(*
  This fb handles mechanical print unit corrections.
  - a 4p grid distortion
  - print unit bar banana correction
  NOTE: temperature extention of whole printbar is still handled in camera
*)
FUNCTION_BLOCK FB_FineAlignement EXTENDS FB_BasePrint IMPLEMENTS I_GridPointCorrection
VAR
  // config
  _fPxResolution     : LREAL; // pixel resolution

  // corrections
  //-- 4 point PU deformation correction/distortion
  //    VISU setup point providing reference and correction (NOTE: persists settings internally)
  _fbPUCorrPoints    : ARRAY[1..4] OF FB_PointCorr;
  //-- banana correction
  _fT1 : LREAL;   // temperature 1
  _fT2 : LREAL;   // temperature 2
  _dx_middle : LREAL;  // correction in middle (for view only)
  _y_max : LREAL; // print unit width [mm]
  //-- PUC 4p correction
  _pAdsCam           : POINTER TO FB_ADS_CAMERA;  // camera interface PUC
  aPucPointNames : ARRAY[1..4] OF STRING := ['1 blue','2 red','3 green','4 olive'];
  
  // helper
  lCtr     : UDINT;
  
  // unit test & debug
  _bUT_4p, _bUT_banana, _bUT_4pPuc : BOOL;
  _sUTPoints_dx : ARRAY[0..nC_UT_cols, 0..nC_UT_rows] OF LREAL;
  _sUTPoints_dy : ARRAY[0..nC_UT_cols, 0..nC_UT_rows] OF LREAL;
  // 4pPUC
  bSelect : ARRAY[1..4] OF BOOL;
  bSelected : ARRAY[1..4] OF BOOL;
  bXPlus, bXMinus, bYPlus, bYMinus : BOOL;
  bTest4pPuc_running : BOOL;
END_VAR
VAR PERSISTENT
  //-- 4point correction
  _bEnable_4p    : BOOL := FALSE;
  _bEnablePuc_4p : BOOL := FALSE;
  //  persistence of points see: FB_PointCorr
  //-- banana correction
  _bEnable_banana : BOOL := FALSE;
  _e_max_per_deltaT : LREAL := 0.01;  // [mm/°C]  TODO: use from config
END_VAR
VAR CONSTANT
  // Unit test configuration
  nC_UT_cols : DINT := 6;   // for test only
  nC_UT_rows : DINT := 5;   // for test only
END_VAR

// cyclic caluclation and view updates
//        NOTE: deformation is happening in updateCorrection() callback

//-- 4p correction
//   visu overrides (limitation rectancular point definition)
_fbPUCorrPoints[3].fX_Ref := _fbPUCorrPoints[1].fX_Ref;
_fbPUCorrPoints[4].fX_Ref := _fbPUCorrPoints[2].fX_Ref;
_fbPUCorrPoints[2].fY_Ref := _fbPUCorrPoints[1].fY_Ref;
_fbPUCorrPoints[4].fY_Ref := _fbPUCorrPoints[3].fY_Ref;
//   update CorrectionPoints view elements
FOR lCtr := 1 TO 4 DO
  _fbPUCorrPoints[lCtr](); 
END_FOR

//-- banana correction
// just calculate the dx in the middle of the PU, just for the VISU
calc_banana_correction(x_pos:=0, y_pos:=_y_max/(2*1000), fT1:=_fT1, fT2:=_fT2, dx_corr=>_dx_middle);
_dx_middle := _dx_middle * 1000; // [m] --> [mm] for visu

// Unit test
IF _bUT_4p THEN _bUT_4p := FALSE; _test_4p(); END_IF
IF _bUT_banana THEN _bUT_banana := FALSE; _test_banana(); END_IF
IF _bUT_4pPuc THEN _test_Puc4p(); END_IF

METHOD PRIVATE _test_4p
VAR
  sPoint : ST_DeformationPoint;
  nCol, nRow, nCrPoint : DINT;
  dx, dy : LREAL;       // correction in [m]
  dx_px, dy_px : DINT;  // correction in [px]
  pPUC_CorrPointsInd : POINTER TO ARRAY[1..4] OF ST_CORRECTION_POINT;
  
  nCorrectionX : ARRAY[1..4] OF REAL := [-0.25, -0.2, 0.35, 0.35];
  nCorrectionY : ARRAY[1..4] OF REAL := [-0.45, -0.3, -0.8, -0.65];
  nCorrectionPointX_PLC : ARRAY[1..4] OF REAL := [0, 1000,   0, 1000];
  nCorrectionPointY_PLC : ARRAY[1..4] OF REAL := [0,   0, 702, 702];
  nCorrectionPointX_PUC : ARRAY[1..4] OF REAL := [0, 671.99,   0, 671.99];
  nCorrectionPointY_PUC : ARRAY[1..4] OF REAL := [-0.0001666666, -0.0001666666, 754.2108, 754.2108];
END_VAR
// setup test correcton points location for PLC & PUC 4p testing
pPUC_CorrPointsInd := _pAdsCam^.pCorrectionPointsIndication;
IF pPUC_CorrPointsInd = 0 THEN F_Report_Error(ErrType:=EN_REPORT_ERROR_TYPE.Report_Error_0Pointer);  RETURN; END_IF

FOR nCrPoint:=1 TO 4 DO
  // correction point location
  // -- PLC
  _fbPUCorrPoints[nCrPoint].fX_Ref := nCorrectionPointX_PLC[nCrPoint];
  _fbPUCorrPoints[nCrPoint].fY_Ref := nCorrectionPointY_PLC[nCrPoint];
  // -- PUC  
  pPUC_CorrPointsInd^[nCrPoint].posx := nCorrectionPointX_PUC[nCrPoint];
  pPUC_CorrPointsInd^[nCrPoint].posy := nCorrectionPointY_PUC[nCrPoint];
  
  // point correction  
  // -- PLC
  _fbPUCorrPoints[nCrPoint].fX := nCorrectionX[nCrPoint];
  _fbPUCorrPoints[nCrPoint].fY := nCorrectionY[nCrPoint];
  // -- PUC
  pPUC_CorrPointsInd^[nCrPoint].x := nCorrectionX[nCrPoint];
  pPUC_CorrPointsInd^[nCrPoint].y := nCorrectionY[nCrPoint];
END_FOR

// generate internal test grid
FOR nCol:=0 TO nC_UT_cols DO
  FOR nRow:=0 TO nC_UT_rows DO
    sPoint.col := nCol;
    sPoint.row := nRow;
    sPoint.x_ref := nCol * TO_DINT(GVL_Deformation.nC_DefaultGridPitch_X);
    sPoint.y_ref := nRow * TO_DINT(GVL_Deformation.nC_DefaultGridPitch_Y);
    sPoint.dx := 0;   // no previous deformation
    sPoint.dy := 0;   // no previous deformation
    
    // calc 4p PLC correction and apply to point
    calc_4p_correction(
        x_pos:=F_SubPixelToMeter(lPosSubPx:=sPoint.x_ref, fResSubPx:=_fPxResolution), 
        y_pos:=F_SubPixelToMeter(lPosSubPx:=sPoint.y_ref, fResSubPx:=_fPxResolution), 
        dx_corr=>dx, 
        dy_corr=>dy);
    LogInfo(
      F_Concat4(
        '4p PLC: point:', 
        F_Concat4(' x=', TO_STRING(sPoint.x_ref), '/y=', TO_STRING(sPoint.y_ref)),
        F_Concat2(' dx=', TO_STRING(dx)),
        F_Concat2(' dy=', TO_STRING(dy))
      )
    );

    // --- store in table for verification with Excel caluculation
    dx_px := F_MeterToSubPixel(fPosMeter:=dx, fResoSubPx:=_fPxResolution);
    dy_px := F_MeterToSubPixel(fPosMeter:=dy, fResoSubPx:=_fPxResolution);
    // save corrected point
    _sUTPoints_dx[nCol, nRow] := dx_px;
    _sUTPoints_dy[nCol, nRow] := dy_px;
    // print corrected point
    LogInfo(
      F_Concat4(
        F_Concat4('[c/r] ', TO_STRING(sPoint.col), '/', TO_STRING(sPoint.row)),
        F_Concat7(' dx: ', TO_STRING(sPoint.dx), '>', TO_STRING(dx_px), ' (', TO_STRING(dx), ')'),
        F_Concat7(' dy: ', TO_STRING(sPoint.dy), '>', TO_STRING(dy_px), ' (', TO_STRING(dy), ')'),
        SEL(sPoint.dx<>dx_px OR sPoint.dy<>dy_px,'',' !!!')
      )
    );
    // ---------------------------------
    
    // calc 4p PUC correction and apply to point
    calc_PUC_4p_correction(
        x_pos:=F_SubPixelToMeter(lPosSubPx:=sPoint.x_ref, fResSubPx:=_fPxResolution), 
        y_pos:=F_SubPixelToMeter(lPosSubPx:=sPoint.y_ref, fResSubPx:=_fPxResolution), 
        dx_corr=>dx, 
        dy_corr=>dy);
    LogInfo(
      F_Concat4(
        '4p PUC: point:', 
        F_Concat4(' x=', TO_STRING(sPoint.x_ref), '/y=', TO_STRING(sPoint.y_ref)),
        F_Concat2(' dx=', TO_STRING(dx)),
        F_Concat2(' dy=', TO_STRING(dy))
      )
    );

  END_FOR  
END_FOR
END_METHOD

METHOD PRIVATE _test_banana
VAR
  sPoint : ST_DeformationPoint;
  nCol, nRow : DINT;
  dx, dy : LREAL;       // correction in [m]
  dx_px, dy_px : LREAL;  // correction in [px]
END_VAR
// generate internal grid
FOR nCol:=0 TO nC_UT_cols DO
  FOR nRow:=0 TO nC_UT_rows DO
    sPoint.col := nCol;
    sPoint.row := nRow;
    sPoint.x_ref := nCol * TO_DINT(GVL_Deformation.nC_DefaultGridPitch_X);
    sPoint.y_ref := nRow * TO_DINT(GVL_Deformation.nC_DefaultGridPitch_Y);
    sPoint.dx := 0;   // no previous deformation
    sPoint.dy := 0;   // no previous deformation
    
    // calc correction and apply to point
    calc_banana_correction(
        x_pos:=F_SubPixelToMeter(lPosSubPx:=sPoint.x_ref, fResSubPx:=_fPxResolution), 
        Y_pos:=F_SubPixelToMeter(lPosSubPx:=sPoint.y_ref, fResSubPx:=_fPxResolution),
        fT1 := 68,
        fT2 := 48, 
        dx_corr=>dx
    );
    dx_px := dx;
    dy_px := dy;
    // save corrected point (dx @y-pos)
    _sUTPoints_dx[nCol, nRow] := dx_px;
    _sUTPoints_dy[nCol, nRow] := F_SubPixelToMeter(lPosSubPx:=sPoint.y_ref, fResSubPx:=_fPxResolution)*1000;
    
    // print corrected point
    LogInfo(
      F_Concat4(
        F_Concat4('[c/r] ', TO_STRING(sPoint.col), '/', TO_STRING(sPoint.row)),
        F_Concat6(' dx: ', TO_STRING(sPoint.dx), '>', TO_STRING(TO_DINT(dx_px)), ' [', TO_STRING(dx)),
        F_Concat6('  dy: ', TO_STRING(sPoint.dy), '>', TO_STRING(TO_DINT(dy_px)), ' [', TO_STRING(dy)),
        SEL(sPoint.dx<>dx_px OR sPoint.dy<>dy_px,'',' !!!')
      )
    );
  END_FOR  
END_FOR
END_METHOD

METHOD PRIVATE _test_Puc4p
VAR
  i : UDINT;

  pPUC_CorrPointsInd : POINTER TO ARRAY[1..4] OF ST_CORRECTION_POINT;
  pPoint : POINTER TO ST_CORRECTION_POINT;
END_VAR
pPUC_CorrPointsInd := _pAdsCam^.pCorrectionPointsIndication;      // get points array from ADS
IF pPUC_CorrPointsInd = 0 THEN F_Report_Error(ErrType:=EN_REPORT_ERROR_TYPE.Report_Error_0Pointer);  RETURN; END_IF

// do selection
IF    bSelect[1] THEN bSelect[1]:=FALSE; MEMSET(destAddr:=ADR(bSelected), fillByte:=0, n:=SIZEOF(bSelected)); bSelected[1] := TRUE;
ELSIF bSelect[2] THEN bSelect[2]:=FALSE; MEMSET(destAddr:=ADR(bSelected), fillByte:=0, n:=SIZEOF(bSelected)); bSelected[2] := TRUE;
ELSIF bSelect[3] THEN bSelect[3]:=FALSE; MEMSET(destAddr:=ADR(bSelected), fillByte:=0, n:=SIZEOF(bSelected)); bSelected[3] := TRUE;
ELSIF bSelect[4] THEN bSelect[4]:=FALSE; MEMSET(destAddr:=ADR(bSelected), fillByte:=0, n:=SIZEOF(bSelected)); bSelected[4] := TRUE;
END_IF

IF    bSelected[1] THEN pPoint := ADR(pPUC_CorrPointsInd^[1]);
ELSIF bSelected[2] THEN pPoint := ADR(pPUC_CorrPointsInd^[2]);
ELSIF bSelected[3] THEN pPoint := ADR(pPUC_CorrPointsInd^[3]);
ELSIF bSelected[4] THEN pPoint := ADR(pPUC_CorrPointsInd^[4]);
ELSE                    pPoint := ADR(pPUC_CorrPointsInd^[1]);
END_IF

IF bXPlus  THEN bXPlus  := FALSE; pPoint^.x := pPoint^.x + 0.05; END_IF
IF bXMinus THEN bXMinus := FALSE; pPoint^.x := pPoint^.x - 0.05; END_IF
IF bYPlus  THEN bYPlus  := FALSE; pPoint^.y := pPoint^.y + 0.05; END_IF
IF bYMinus THEN bYMinus := FALSE; pPoint^.y := pPoint^.y - 0.05; END_IF
END_METHOD

(*
  Calculate grid point displacement for a distortion with 4 rectangular defined points.
  Uses 2-bilinear interpolation between the 4 rectancular reference points.
*)
METHOD PRIVATE calc_4p_correction : BOOL
VAR_INPUT
  x_pos   : LREAL;    // point x position [m]
  y_pos   : LREAL;    // point y position [m]
END_VAR
VAR_OUTPUT
  dx_corr : LREAL;    // point correction x [m]
  dy_corr : LREAL;    // point correction y [m]
END_VAR
VAR
  dx, dy : LREAL;     // difference between Calibration Points (rectangle)
  x1, x2, y1, y2 : LREAL;
  cx1, cx2, cy1, cy2 : LREAL;
  GPx, GPy : LREAL;
  CVx, CVy : LREAL;
  lErrCtr : UDINT;
END_VAR

// Grid point position
GPx := x_pos; 
GPy := y_pos;

// Interpolation in x
x1 := _fbPUCorrPoints[1].fX_Ref / 1000;    // [mm -> m]
x2 := _fbPUCorrPoints[2].fX_Ref / 1000;    // [mm -> m]
dx := x2-x1;
IF dx = 0 THEN (*F_Report_Error(ErrType:=EN_REPORT_ERROR_TYPE.Report_Error_0Pointer);*) RETURN; END_IF

cx1 := (x2-GPx)/dx * (_fbPUCorrPoints[1].fX / 1000) + (GPx-x1)/dx * (_fbPUCorrPoints[2].fX / 1000);
cx2 := (x2-GPx)/dx * (_fbPUCorrPoints[3].fX / 1000) + (GPx-x1)/dx * (_fbPUCorrPoints[4].fX / 1000);
cy1 := (x2-GPx)/dx * (_fbPUCorrPoints[1].fY / 1000) + (GPx-x1)/dx * (_fbPUCorrPoints[2].fY / 1000);
cy2 := (x2-GPx)/dx * (_fbPUCorrPoints[3].fY / 1000) + (GPx-x1)/dx * (_fbPUCorrPoints[4].fY / 1000);

// Interpolation in y
y1 := _fbPUCorrPoints[1].fY_Ref / 1000;    // [mm -> m]
y2 := _fbPUCorrPoints[3].fY_Ref / 1000;    // [mm -> m]
dy := y2-y1;
IF dy = 0 THEN (*F_Report_Error(ErrType:=EN_REPORT_ERROR_TYPE.Report_Error_0Pointer);*) RETURN; END_IF

// Calc interpolated 
CVx := (y2 - GPy)/dy * cx1 + (GPy-y1)/dy * cx2;
CVy := (y2 - GPy)/dy * cy1 + (GPy-y1)/dy * cy2;

// return accurate new correction only
dx_corr := CVx;
dy_corr := CVy;

calc_4p_correction := TRUE;
END_METHOD

(*
  Calculate grid point displacement for print unit banana deformation.
  2nd order approximation.
*)
METHOD PRIVATE calc_banana_correction : BOOL
VAR_INPUT
  x_pos   : LREAL;    // point x position [m]
  y_pos   : LREAL;    // point y position [m]
  fT1     : LREAL;    // temperature 1 [°C]
  fT2     : LREAL;    // temperature 2 [°C]
END_VAR
VAR_OUTPUT
  dx_corr : LREAL;    // point correction x [m]
END_VAR
VAR
  delta_T : LREAL;   // delta temperature
  e_max   : LREAL;   //
  a : LREAL;
  x_dash, y_dash : LREAL;
END_VAR
IF _y_max = 0 THEN RETURN; END_IF

x_dash := y_pos * 1000; // [m] -> [mm]

delta_T := fT2-fT1;
e_max   := delta_T * _e_max_per_deltaT;

a := 4 * e_max /  EXPT(_y_max, 2);
y_dash := a * EXPT(x_dash - (_y_max / 2), 2) - e_max;

// correction value
dx_corr := (y_dash / 1000);  // [mm] -> [m]

calc_banana_correction := TRUE;
END_METHOD

(*
  Calculate grid point displacement for a distortion with 4 rectangular defined points.
  Uses 2-bilinear interpolation between the 4 rectancular reference points.
*)
METHOD PRIVATE calc_PUC_4p_correction : BOOL
VAR_INPUT
  x_pos   : LREAL;    // point x position [m]
  y_pos   : LREAL;    // point y position [m]
END_VAR
VAR_OUTPUT
  dx_corr : LREAL;    // point correction x [m]
  dy_corr : LREAL;    // point correction y [m]
END_VAR
VAR
  dx, dy : LREAL;     // difference between Calibration Points (rectangle)
  x1, x2, y1, y2 : LREAL;
  cx1, cx2, cy1, cy2 : LREAL;
  GPx, GPy : LREAL;
  CVx, CVy : LREAL;
  lErrCtr : UDINT;
  
  pPUC_CorrPointsInd : POINTER TO ARRAY[1..4] OF ST_CORRECTION_POINT;
END_VAR
VAR CONSTANT
  bC_InvertValX : BOOL := TRUE;
  bC_InvertValY : BOOL := FALSE;
END_VAR
pPUC_CorrPointsInd := _pAdsCam^.pCorrectionPointsIndication;      // get points array from ADS
IF pPUC_CorrPointsInd = 0 THEN F_Report_Error(ErrType:=EN_REPORT_ERROR_TYPE.Report_Error_0Pointer);  RETURN; END_IF

// Grid point position
GPx := x_pos; 
GPy := y_pos;

// Interpolation in x
x1 := pPUC_CorrPointsInd^[1].posx / 1000;    // [mm -> m]
x2 := pPUC_CorrPointsInd^[2].posx / 1000;    // [mm -> m]
dx := x2-x1;
IF dx = 0 THEN (*F_Report_Error(ErrType:=EN_REPORT_ERROR_TYPE.Report_Error_0Pointer);*) RETURN; END_IF

// NOTE: x is inverted (compare to fX / fY method of FB_PointCorr)
cx1 := (x2-GPx)/dx * ((pPUC_CorrPointsInd^[1].x * -1) / 1000) + (GPx-x1)/dx * ((pPUC_CorrPointsInd^[2].x * -1) / 1000);
cx2 := (x2-GPx)/dx * ((pPUC_CorrPointsInd^[3].x * -1) / 1000) + (GPx-x1)/dx * ((pPUC_CorrPointsInd^[4].x * -1) / 1000);
cy1 := (x2-GPx)/dx * ((pPUC_CorrPointsInd^[1].y) / 1000) + (GPx-x1)/dx * ((pPUC_CorrPointsInd^[2].y) / 1000);
cy2 := (x2-GPx)/dx * ((pPUC_CorrPointsInd^[3].y) / 1000) + (GPx-x1)/dx * ((pPUC_CorrPointsInd^[4].y) / 1000);

// Interpolation in y
y1 := pPUC_CorrPointsInd^[1].posy / 1000;    // [mm -> m]
y2 := pPUC_CorrPointsInd^[3].posy / 1000;    // [mm -> m]
dy := y2-y1;
IF dy = 0 THEN (*F_Report_Error(ErrType:=EN_REPORT_ERROR_TYPE.Report_Error_0Pointer);*) RETURN; END_IF

// Calc interpolated 
CVx := (y2 - GPy)/dy * cx1 + (GPy-y1)/dy * cx2;
CVy := (y2 - GPy)/dy * cy1 + (GPy-y1)/dy * cy2;

// return accurate new correction only
dx_corr := CVx;
dy_corr := CVy;

calc_PUC_4p_correction := TRUE;
END_METHOD

PROPERTY fT_PL1 : LREAL
SET
_fT1 := fT_PL1;
END_SET
END_PROPERTY

PROPERTY fT_PL2 : LREAL
SET
_fT2 := fT_PL2;
END_SET
END_PROPERTY

METHOD init : BOOL
VAR_INPUT
  pAdsCam        : POINTER TO FB_ADS_CAMERA;  // camera interface PUC
  fPxReso        : LREAL;   // pixel resolution
  fPuWidth       : LREAL;   // Print unit width [m]
END_VAR
_fPxResolution := fPxReso;
_y_max         := fPuWidth * 1000;  // -> [mm]
_pAdsCam       := pAdsCam;
IF _pAdsCam = 0 THEN LogError('missing _pAdsCam, ads interface unknown, call worker specific init before'); END_IF

// PU Deformation
_fbPUCorrPoints[1].init(aName:='P1', aUnit:='mm', fX_Min:=-5, fX_Max:=5, fY_Min:=-5, fY_Max:=5, fIncrStep:=0.05, 
                        bButnInvertX:=TRUE, bButnInvertY:=TRUE, bValInvertX:=TRUE, bValInvertY:=FALSE);
_fbPUCorrPoints[2].init(aName:='P2', aUnit:='mm', fX_Min:=-5, fX_Max:=5, fY_Min:=-5, fY_Max:=5, fIncrStep:=0.05,
                        bButnInvertX:=TRUE, bButnInvertY:=TRUE, bValInvertX:=TRUE, bValInvertY:=FALSE);
_fbPUCorrPoints[3].init(aName:='P3', aUnit:='mm', fX_Min:=-5, fX_Max:=5, fY_Min:=-5, fY_Max:=5, fIncrStep:=0.05,
                        bButnInvertX:=TRUE, bButnInvertY:=TRUE, bValInvertX:=TRUE, bValInvertY:=FALSE);
_fbPUCorrPoints[4].init(aName:='P4', aUnit:='mm', fX_Min:=-5, fX_Max:=5, fY_Min:=-5, fY_Max:=5, fIncrStep:=0.05,
                        bButnInvertX:=TRUE, bButnInvertY:=TRUE, bValInvertX:=TRUE, bValInvertY:=FALSE);
END_METHOD

(*
  Apply fine-alignement corrections to DefGrid point
*)
METHOD updateCorrection : BOOL
VAR_INPUT
  pPoint : POINTER TO ST_DeformationPointAccurate;
END_VAR
VAR
  x_pos, dx_corr, dx_tmp : LREAL; // [m]
  y_pos, dy_corr, dy_tmp : LREAL; // [m]
END_VAR
// grid point position
x_pos := F_SubPixelToMeter(lPosSubPx:=FC_LREAL_TO_DINT(pPoint^.x_ref), fResSubPx:=_fPxResolution);  // [px -> m] 
y_pos := F_SubPixelToMeter(lPosSubPx:=FC_LREAL_TO_DINT(pPoint^.y_ref), fResSubPx:=_fPxResolution);  // [px -> m]
dx_corr := 0;
dy_corr := 0;

// calc - 4 point sheet deformation (PU and machine mechanical distortions)
IF _bEnable_4p THEN
  calc_4p_correction(x_pos:=x_pos, y_pos:=y_pos, dx_corr=>dx_tmp, dy_corr=>dy_tmp);
  dx_corr := dx_tmp + dx_corr;
  dy_corr := dy_tmp + dy_corr;
END_IF

IF _bEnablePuc_4p THEN  (*PUC 4P correction used*)
  calc_PUC_4p_correction(x_pos:=x_pos, y_pos:=y_pos, dx_corr=>dx_tmp, dy_corr=>dy_tmp);
  dx_corr := dx_tmp + dx_corr;
  dy_corr := dy_tmp + dy_corr;
END_IF

// calc - banana correction
IF _bEnable_banana THEN
  calc_banana_correction(x_pos:=x_pos, y_pos:=y_pos, fT1:=_fT1, fT2:=_fT2, dx_corr=>dx_tmp);
  dx_corr := dx_tmp + dx_corr;
END_IF
// apply new correction to deformation correction 
pPoint^.dx := pPoint^.dx + F_MeterToSubPixelReal(fPosMeter:=dx_corr, fResoSubPx:=_fPxResolution);
pPoint^.dy := pPoint^.dy + F_MeterToSubPixelReal(fPosMeter:=dy_corr, fResoSubPx:=_fPxResolution);

updateCorrection := TRUE;
END_METHOD

END_FUNCTION_BLOCK

(* stored: Version 1.1.0.1, ProductVersion 3.1.4024.11
   POU FB_FineAlignement: Id {b0fdbfcd-2a71-4ede-b938-0e28dbf7b80d}, SpecialFunc None
   Method _test_4p: Id {6f0fa0b6-cc58-4465-bff5-26ae640a97c0}
   Method _test_banana: Id {cdda5b50-a20e-4ef0-8e55-027af444ef1f}
   Method _test_Puc4p: Id {1465faa5-e93a-4ecc-a1a2-9fc2ea753518}
   Method calc_4p_correction: Id {c5b8318f-9300-4b60-afbb-0f066a2ad2b7}
   Method calc_banana_correction: Id {cd11fc31-cdd1-4fff-a3a1-69aafb3db5bd}
   Method calc_PUC_4p_correction: Id {49285f29-32e6-41ef-a994-fe07d41d686f}
   Property fT_PL1: Id {b286c81c-0aff-4511-94c9-d4cc9bd4439b}
   Set Set: Id {c98c4823-db0a-4cb5-8e5c-1cb8271580d0}
   Property fT_PL2: Id {54ff08d7-dae5-4a96-a73a-97aa019a8e38}
   Set Set: Id {1684f327-46b0-49b3-a6db-fbee77699606}
   Method init: Id {22d51a6a-e008-40d7-a511-92f228aee50f}
   Method updateCorrection: Id {67567b6c-ad9f-4c43-b042-ce1ae67d99c3} *)
